// TwinCAT 3 PLC project PLC
// ProgramVersion: 3.1.4024.12
// libraries:
//   Tc2_Standard, * (Beckhoff Automation GmbH)
//   Tc2_System, * (Beckhoff Automation GmbH)
//   Tc3_Module, * (Beckhoff Automation GmbH)
//   Util, * (System)
// project tree:
//   DUTs/ DUT.TcDUT
//   GVLs/ GVL.TcGVL, GVL_1.TcGVL
//   / PlcTask.TcTTO
//   POUs/ MAIN.TcPOU

CONFIGURATION PLC
    RESOURCE PLC ON TwinCAT3
        TASK PlcTask(INTERVAL := T#10ms, PRIORITY := 20);
        PROGRAM MAIN WITH PlcTask : MAIN;
    END_RESOURCE
END_CONFIGURATION

// ---- DUTs/DUT.TcDUT
TYPE DUT :
STRUCT
	cc:BOOL;
	dd:INT;
END_STRUCT
END_TYPE

// ---- GVLs/GVL.TcGVL
{attribute 'qualified_only'}
VAR_GLOBAL
	g:BOOL;
END_VAR

// ---- GVLs/GVL_1.TcGVL
{attribute 'qualified_only'}
VAR_GLOBAL
END_VAR

// ---- POUs/MAIN.TcPOU
PROGRAM MAIN
VAR
	a:BOOL;
	b:INT;
	dut:DUT;
END_VAR

a:=TRUE;
b:=11;
GVL.g:=TRUE;
dut.cc:=FALSE;

END_PROGRAM
